Fanuc KAREL source: kt00376.compact.KL

PROGRAM KT00376
%STACKSIZE=65535
%PRIORITY=65535
%NOLOCKGROUP
VAR
Y1 : ARRAY[2] OF BYTE
R2 : REAL
OUT : BOOLEAN
BEGIN
Y1[1]=2
R2=3.0
OUT=((Y1[1]) <=R2)
END KT00376
